FUNCTION_BLOCK AnalogMultiplexer
VAR_INPUT
	bSelect: BOOL;
	iSelect: INT := -1;
	In0: LREAL := 0;
	In1: LREAL := 0;
	In2: LREAL := 0;
	In3: LREAL := 0;
END_VAR
VAR_OUTPUT
	Out: LREAL;
END_VAR
VAR
END_VAR

IF iSelect = -1 THEN
	IF bSelect THEN
		Out := In1;
	ELSE
		Out := In0;
	END_IF
ELSE
	CASE iSelect OF
		0: 	Out := In0;
		1: 	Out := In1;
		2: 	Out := In2;
		3: 	Out := In3;
	END_CASE
END_IF

END_FUNCTION_BLOCK

(* stored: Version 1.1.0.1, ProductVersion 3.1.4024.3
   POU AnalogMultiplexer: Id {a7e760a3-8baa-4cca-8e27-694b8ef3f927}, SpecialFunc None *)
